TYPE AdsTagsSmokeControl :
STRUCT
	Status: GreenMasterStatusSmokeControl;
END_STRUCT
END_TYPE

(* stored: Version 1.1.0.1, ProductVersion 3.1.4024.6
   DUT AdsTagsSmokeControl: Id {ef66e122-5258-4237-a330-ce75163ffe21} *)
